(* PLC project v0.6.02_RefactorGateAndTest.project, CODESYS CODESYS V3.5 SP19 Patch 1 *)
(* stored: creationDateTime 2026-07-27T19:30:23.027286, modificationDateTime 2026-07-27T19:30:23.027286 *)

TYPE ST_WinchSymmetryHMI : STRUCT
  BtnReset : BOOL;
  SymmetryOk : BOOL;
  SymmetryValid : BOOL;
  DeltaStartDelay_Ms : UDINT;
  DeltaBrakeReleaseTime_Ms : UDINT;
  DeltaBrakeApplyTime_Ms : UDINT;
  DeltaStopDistance_M : REAL;
  DeltaStopTime_Ms : UDINT;
  MaxSyncDeviation_M : REAL;
END_STRUCT;
END_TYPE
